// TIA Portal V19 export
FUNCTION_BLOCK "SafetyZone1Actuators"   // FB113, F_LAD
// In this function block, the actuator control is implemented.
// stored: IsIECCheckEnabled true, Namespace Safety
   VAR_INPUT
      ack { ExternalWritable := 'False'} : Bool;   // Acknowledge
      release { ExternalWritable := 'False'} : Bool;   // Relese all safety
      statusWordDrive1 { ExternalWritable := 'False'} : "Safety.LDrvSafe_typeSinaSTlg30Status";
      statusWordDrive2 { ExternalWritable := 'False'} : "Safety.LDrvSafe_typeSinaSTlg30Status";
   END_VAR
   VAR_OUTPUT
      ackReq { ExternalWritable := 'False'} : Bool;   // Acknowledge required
      safetyFault { ExternalWritable := 'False'} : Bool;   // Safety Fault active
      stoActive { ExternalWritable := 'False'} : Bool;   // STO active
      statusDrive1 { ExternalWritable := 'False'} : "Safety.typeSafetyDrive";
      statusDrive2 { ExternalWritable := 'False'} : "Safety.typeSafetyDrive";
      controlWordDrive1 { ExternalWritable := 'False'} : "Safety.LDrvSafe_typeSinaSTlg30Control";
      controlWordDrive2 { ExternalWritable := 'False'} : "Safety.LDrvSafe_typeSinaSTlg30Control";
   END_VAR
   VAR
      instContactor { ExternalWritable := 'False'} : FDBACK;   // Status feedback of the actuator
      instDrive1 { ExternalWritable := 'False'} : "Safety.DrvSafeSinaSTlg30";
      instDrive2 { ExternalWritable := 'False'} : "Safety.DrvSafeSinaSTlg30";
   END_VAR
BEGIN

REGION Network 1: Switch contactor
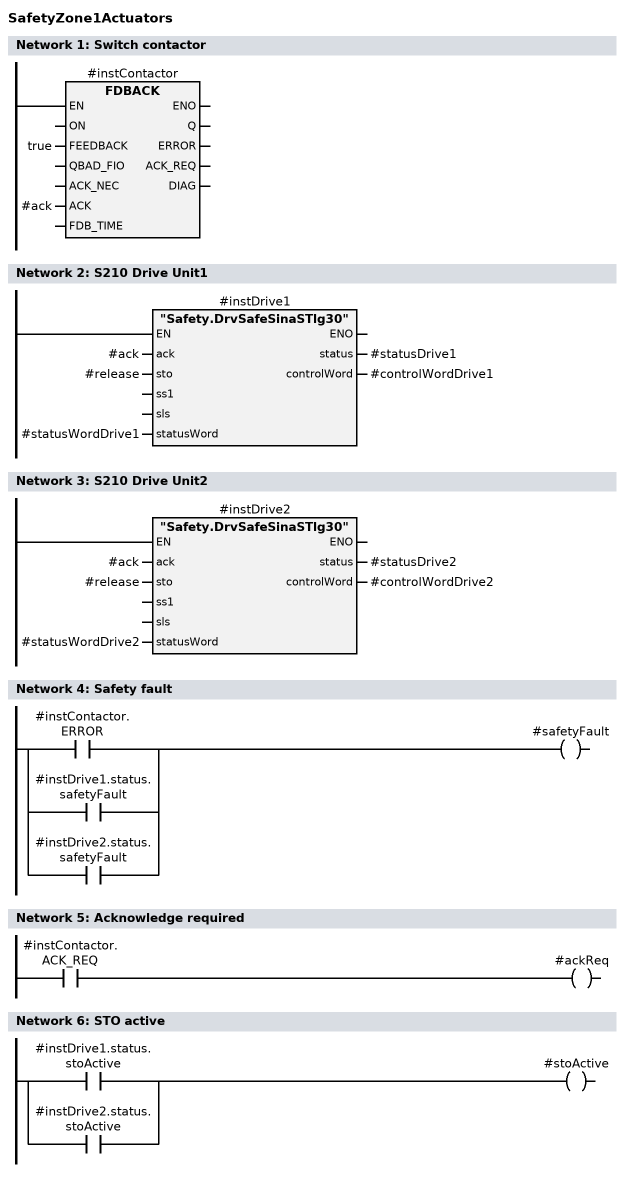
   RUNG wire#powerrail
      #instContactor.FDBACK(ON :=, FEEDBACK := true, QBAD_FIO :=, ACK_NEC :=, ACK := #ack, FDB_TIME :=, Q =>, ERROR =>, ACK_REQ =>, DIAG =>)
   END_RUNG
   // the same network as SCL:
   #instContactor(FEEDBACK := true, ACK := #ack);   // FDBACK
END_REGION

REGION Network 2: S210 Drive Unit1
   RUNG wire#powerrail
      #instDrive1(ack := #ack, sto := #release, ss1 :=, sls :=, statusWord := #statusWordDrive1, status => #statusDrive1, controlWord => #controlWordDrive1)
   END_RUNG
   // the same network as SCL:
   #instDrive1(ack := #ack,   // "Safety.DrvSafeSinaSTlg30"
               sto := #release,
               statusWord := #statusWordDrive1,
               status => #statusDrive1,
               controlWord => #controlWordDrive1);
END_REGION

REGION Network 3: S210 Drive Unit2
   RUNG wire#powerrail
      #instDrive2(ack := #ack, sto := #release, ss1 :=, sls :=, statusWord := #statusWordDrive2, status => #statusDrive2, controlWord => #controlWordDrive2)
   END_RUNG
   // the same network as SCL:
   #instDrive2(ack := #ack,   // "Safety.DrvSafeSinaSTlg30"
               sto := #release,
               statusWord := #statusWordDrive2,
               status => #statusDrive2,
               controlWord => #controlWordDrive2);
END_REGION

REGION Network 4: Safety fault
   RUNG wire#powerrail
      Contact( #instContactor.ERROR )
      wire#w1
      Coil( #safetyFault )
   END_RUNG
   RUNG wire#powerrail
      Contact( #instDrive1.status.safetyFault )
   END_RUNG wire#w1
   RUNG wire#powerrail
      Contact( #instDrive2.status.safetyFault )
   END_RUNG wire#w1
   // the same network as SCL:
   #safetyFault := #instContactor.ERROR OR #instDrive1.status.safetyFault OR #instDrive2.status.safetyFault;
END_REGION

REGION Network 5: Acknowledge required
   RUNG wire#powerrail
      Contact( #instContactor.ACK_REQ )
      Coil( #ackReq )
   END_RUNG
   // the same network as SCL:
   #ackReq := #instContactor.ACK_REQ;
END_REGION

REGION Network 6: STO active
   RUNG wire#powerrail
      Contact( #instDrive1.status.stoActive )
      wire#w1
      Coil( #stoActive )
   END_RUNG
   RUNG wire#powerrail
      Contact( #instDrive2.status.stoActive )
   END_RUNG wire#w1
   // the same network as SCL:
   #stoActive := #instDrive1.status.stoActive OR #instDrive2.status.stoActive;
END_REGION
END_FUNCTION_BLOCK
